TYPE IPC :
STRUCT
		
		MesAlarmCode		: WORD ;	(* (NA) Internal Akuo AlarmCode		*)
		MesWarningCode		: WORD ; 	(* (NA) Internal Akuo WarningCode   *)
		MesEventCode		: WORD ; 	(* (NA) Internal Akuo EventCode	    *)
		
END_STRUCT
END_TYPE

(* stored: Version 1.1.0.1, ProductVersion 3.1.4024.6
   DUT IPC: Id {c9f97eda-b976-4b6e-baea-497eca27c656} *)
